(* IEC 61131-3 sources: RL_MAR/experiments/comparison/llm4plc/results/deepseek-ai-DeepSeek-V3.2_20260506_104945/20260506_110926, 1 file *)

(* ---- generated_code_iteration_0.st ---- *)
START_ST
FUNCTION_BLOCK FB_BottleProcessing
VAR_INPUT
    bottleSensor : BOOL;
    cleaningConfirmButton : BOOL;
    fillingConfirmButton : BOOL;
    cappingConfirmButton : BOOL;
    packingConfirmButton : BOOL;
    finishedButton : BOOL;
END_VAR

VAR_OUTPUT
    Pump_Motor : BOOL;
    Filling_Valve : BOOL;
    Capping_Machine : BOOL;
    Packing_Machine : BOOL;
    Completion_Light : BOOL;
END_VAR

VAR
    State : INT := 0;
END_VAR

CASE State OF
    0: (* WAITING *)
        Pump_Motor := FALSE;
        Filling_Valve := FALSE;
        Capping_Machine := FALSE;
        Packing_Machine := FALSE;
        Completion_Light := FALSE;
        IF bottleSensor THEN
            Pump_Motor := TRUE;
            State := 1;
        END_IF;

    1: (* CLEANING *)
        Pump_Motor := TRUE;
        Filling_Valve := FALSE;
        Capping_Machine := FALSE;
        Packing_Machine := FALSE;
        Completion_Light := FALSE;
        IF cleaningConfirmButton THEN
            Pump_Motor := FALSE;
            Filling_Valve := TRUE;
            State := 2;
        END_IF;

    2: (* FILLING *)
        Pump_Motor := FALSE;
        Filling_Valve := TRUE;
        Capping_Machine := FALSE;
        Packing_Machine := FALSE;
        Completion_Light := FALSE;
        IF fillingConfirmButton THEN
            Filling_Valve := FALSE;
            Capping_Machine := TRUE;
            State := 3;
        END_IF;

    3: (* CAPPING *)
        Pump_Motor := FALSE;
        Filling_Valve := FALSE;
        Capping_Machine := TRUE;
        Packing_Machine := FALSE;
        Completion_Light := FALSE;
        IF cappingConfirmButton THEN
            Capping_Machine := FALSE;
            Packing_Machine := TRUE;
            State := 4;
        END_IF;

    4: (* PACKING *)
        Pump_Motor := FALSE;
        Filling_Valve := FALSE;
        Capping_Machine := FALSE;
        Packing_Machine := TRUE;
        Completion_Light := FALSE;
        IF packingConfirmButton THEN
            Packing_Machine := FALSE;
            Completion_Light := TRUE;
            State := 5;
        END_IF;

    5: (* COMPLETED *)
        Pump_Motor := FALSE;
        Filling_Valve := FALSE;
        Capping_Machine := FALSE;
        Packing_Machine := FALSE;
        Completion_Light := TRUE;
        IF finishedButton THEN
            Completion_Light := FALSE;
            State := 0;
        END_IF;
END_CASE;
END_FUNCTION_BLOCK
END_ST
